# EPICS substitutions: pmacApp/Db/pmac.substitutions
# This file was automatically generated on Thu 15 Nov 2018 14:28:58 GMT from
# source: /home/hgv27681/R3.14.12.7/support/pmac/etc/makeIocs/lab.xml
#
# *** Please do not edit this file: edit the source file instead. ***
#

# Macros:
#  PORT      The asyn port for the pmac controller
#  P         PV Prefix
#  NAXES     Number of axes
#  TIMEOUT   Timeout for controller communication
#  FEEDRATE  feedrate below which we go into error
#  CSG0      Name for Coordinate System Group 0
#  CSG1      Name for Coordinate System Group 1
#  CSG2      Name for Coordinate System Group 2
#  CSG3      Name for Coordinate System Group 3
#  CSG4      Name for Coordinate System Group 4
#  CSG5      Name for Coordinate System Group 5
#  CSG6      Name for Coordinate System Group 6
#  CSG7      Name for Coordinate System Group 7
#file /usr/local/epics-nfs/apps/pmac/2019_05_14_01/db/pmacController.template
file /usr/local/epics-nfs/apps/pmac/pmacApp/Db/pmacController.template
{
pattern { PORT, P, NAXES, TIMEOUT, FEEDRATE, CSG0, CSG1, CSG2, CSG3, CSG4, CSG5, CSG6, CSG7 }
    { "Brick", "BRICK1", "8", "4", "100", "", "", "", "", "", "", "", "" }
}

# Macros:
#  PORT  The asyn port for the pmac controller
#  P     PV Prefix
#file /usr/local/epics-nfs/apps/pmac/2019_05_14_01/db/powerPmacStatus.template
file /usr/local/epics-nfs/apps/pmac/pmacApp/Db/powerPmacStatus.template
{
pattern { PORT, P }
    { "Brick", "BRICK1" }
}

# Macros:
#  PMAC  Pmac/Geobrick name
#  AXIS  Axis number
#  PORT  Asyn port
#file /usr/local/epics-nfs/apps/pmac/2019_05_14_01/db/pmacStatusAxis.template
file /usr/local/epics-nfs/apps/pmac/pmacApp/Db/pmacStatusAxis.template
{
pattern { PMAC, AXIS, PORT }
    { "BRICK1", "1", "Brick" }
    { "BRICK1", "2", "Brick" }
    { "BRICK1", "3", "Brick" }
    { "BRICK1", "4", "Brick" }
    { "BRICK1", "5", "Brick" }
    { "BRICK1", "6", "Brick" }
    { "BRICK1", "7", "Brick" }
    { "BRICK1", "8", "Brick" }
}

#file /usr/local/epics-nfs/apps/pmac/2019_05_14_01/db/pmacCsController.template
#{
#pattern {PORT, PARENTPORT, TIMEOUT, PMAC, CS}
#	{"CS1", "Brick", 100, "BRICK1", 1}
#}

# Macros:
#  P           Device Prefix
#  M           Device Suffix
#  PORT        Delta tau motor CS
#  ADDR        Address on controller
#  DESC        Description, displayed on EDM screen
#  MRES        Motor Step Size (EGU)
#  VELO        Velocity (EGU/s)
#  PREC        Display Precision
#  EGU         Engineering Units
#  TWV         Tweak Step Size (EGU)
#  DTYP        DTYP of record
#  DIR         User Direction
#  VBAS        Base Velocity (EGU/s)
#  VMAX        Max Velocity (EGU/s), defaults to VELO
#  ACCL        Seconds to Velocity
#  BDST        BL Distance (EGU)
#  BVEL        BL Velocity (EGU/s)
#  BACC        BL Seconds to Veloc.
#  DHLM        Dial High Limit
#  DLLM        Dial Low Limit
#  HLM         User High Limit
#  LLM         User Low Limit
#  HLSV        HW Lim. Violation Svr
#  INIT        Startup commands
#  SREV        Steps per Revolution
#  RRES        Readback Step Size (EGU)
#  ERES        Encoder Step Size (EGU)
#  JAR         Jog Acceleration (EGU/s^2)
#  UEIP        Use Encoder If Present
#  URIP        Use RDBL If Present
#  RDBL        Readback Location, set URIP = 1 if you specify this
#  RTRY        Max retry count
#  DLY         Readback settle time (s)
#  OFF         User Offset (EGU)
#  RDBD        Retry Deadband (EGU)
#  FOFF        Freeze Offset, 0=variable, 1=frozen
#  ADEL        Alarm monitor deadband (EGU)
#  NTM         New Target Monitor, only set to 0 for soft motors
#  FEHIGH      HIGH limit for following error
#  FEHIHI      HIHI limit for following error
#  FEHHSV      HIHI alarm severity for following error
#  FEHSV       HIGH alarm severity for following error
#  SCALE       Scale factor, if pmacSetAxisScale is used this should be set
#  HOMEVIS     If 1 then home is visible on the gui
#  HOMEVISSTR  If HOMEVIS=0, then display this text on the gui instead
#  name        Object name and gui association name
#  alh         Set this to alh to add the motor to the alarm handler and send emails,
#  gda_name    Name to export this as to GDA
#  gda_desc    Description to export this as to GDA
#  HOME        Prefix for autohome instance. Defaults to $(P). If unspecified,
#file /usr/local/epics-nfs/apps/pmac/2019_05_14_01/db/dls_pmac_cs_asyn_motor.template
file /usr/local/epics-nfs/apps/pmac/pmacApp/Db/dls_pmac_cs_asyn_motor.template
{
pattern { P, M, PORT, ADDR, DESC, MRES, VELO, PREC, EGU, TWV, DTYP, DIR, VBAS, VMAX, ACCL, BDST, BVEL, BACC, DHLM, DLLM, HLM, LLM, HLSV, INIT, SREV, RRES, ERES, JAR, UEIP, URIP, RDBL, RTRY, DLY, OFF, RDBD, FOFF, ADEL, NTM, FEHIGH, FEHIHI, FEHHSV, FEHSV, SCALE, HOMEVIS, HOMEVISSTR, name, alh, gda_name, gda_desc, HOME, PMAC, CS }
  { "BL", ":vm1", "CS1", "1", "Test motor", "1", "100", "3", "mm", "0.0", "asynMotor", "0", "0", "1000", "0.5", "0", "0", "", "", "", "", "", "MAJOR", "", "1000", "", "", "", "0", "0", "", "0", "0", "0", "", "0", "0", "1", "0", "0", "NO_ALARM", "NO_ALARM", "1", "1", "Use motor summary screen", "BRICK1.MOTORS.M1", "None", "", "Test", "$(P)", "BRICK1", "1" }
  { "BL", ":vm2", "CS1", "2", "Test motor", "1", "100", "3", "mm", "0.0", "asynMotor", "0", "0", "1000", "0.5", "0", "0", "", "", "", "", "", "MAJOR", "", "1000", "", "", "", "0", "0", "", "0", "0", "0", "", "0", "0", "1", "0", "0", "NO_ALARM", "NO_ALARM", "1", "1", "Use motor summary screen", "BRICK1.MOTORS.M2", "None", "", "Test", "$(P)", "BRICK1", "1" }
  { "BL", ":vm3", "CS1", "3", "Test motor", "1", "100", "3", "mm", "0.0", "asynMotor", "0", "0", "1000", "0.5", "0", "0", "", "", "", "", "", "MAJOR", "", "1000", "", "", "", "0", "0", "", "0", "0", "0", "", "0", "0", "1", "0", "0", "NO_ALARM", "NO_ALARM", "1", "1", "Use motor summary screen", "BRICK1.MOTORS.M3", "None", "", "Test", "$(P)", "BRICK1", "1" }
  { "BL", ":vm5", "CS1", "5", "Test motor", "1", "100", "3", "mm", "0.0", "asynMotor", "0", "0", "1000", "0.5", "0", "0", "", "", "", "", "", "MAJOR", "", "1000", "", "", "", "0", "0", "", "0", "0", "0", "", "0", "0", "1", "0", "0", "NO_ALARM", "NO_ALARM", "1", "1", "Use motor summary screen", "BRICK1.MOTORS.M5", "None", "", "Test", "$(P)", "BRICK1", "1" }
  { "BL", ":vm6", "CS1", "6", "Test motor", "1", "100", "3", "mm", "0.0", "asynMotor", "0", "0", "1000", "0.5", "0", "0", "", "", "", "", "", "MAJOR", "", "1000", "", "", "", "0", "0", "", "0", "0", "0", "", "0", "0", "1", "0", "0", "NO_ALARM", "NO_ALARM", "1", "1", "Use motor summary screen", "BRICK1.MOTORS.M6", "None", "", "Test", "$(P)", "BRICK1", "1" }
  { "BL", ":Gap", "CS1", "7", "Horizontal gap", "0.048828125", "10", "3", "um", "0.0", "asynMotor", "0", "0", "1000", "0.5", "0", "0", "", "10000", "-10000", "10000", "-10000", "MAJOR", "", "8192", "", "", "", "0", "0", "", "0", "0", "0", "", "0", "0", "1", "0", "0", "NO_ALARM", "NO_ALARM", "1", "1", "Use motor summary screen", "BRICK1.MOTORS.M7", "None", "", "Test", "$(P)", "BRICK1", "1" }
  { "BL", ":Offset", "CS1", "8", "Horizontal offset", "0.048828125", "10", "3", "um", "0.0", "asynMotor", "0", "0", "1000", "0.5", "0", "0", "", "10000", "-10000", "10000", "-10000", "MAJOR", "", "8192", "", "", "", "0", "0", "", "0", "0", "0", "", "0", "0", "1", "0", "0", "NO_ALARM", "NO_ALARM", "1", "1", "Use motor summary screen", "BRICK1.MOTORS.M8", "None", "", "Test", "$(P)", "BRICK1", "1" }
  { "BL", ":Gap", "CS2", "7", "Vertical gap", "0.048828125", "10", "3", "um", "0.0", "asynMotor", "0", "0", "1000", "0.5", "0", "0", "", "10000", "-10000", "10000", "-10000", "MAJOR", "", "8192", "", "", "", "0", "0", "", "0", "0", "0", "", "0", "0", "1", "0", "0", "NO_ALARM", "NO_ALARM", "1", "1", "Use motor summary screen", "BRICK1.MOTORS.M7", "None", "", "Test", "$(P)", "BRICK1", "2" }
  { "BL", ":Offset", "CS2", "8", "Vertical offset", "0.048828125", "10", "3", "um", "0.0", "asynMotor", "0", "0", "1000", "0.5", "0", "0", "", "10000", "-10000", "10000", "-10000", "MAJOR", "", "8192", "", "", "", "0", "0", "", "0", "0", "0", "", "0", "0", "1", "0", "0", "NO_ALARM", "NO_ALARM", "1", "1", "Use motor summary screen", "BRICK1.MOTORS.M8", "None", "", "Test", "$(P)", "BRICK1", "2" }
}

# Macros:
#  P                Device Prefix
#  M                Device Suffix
#  PORT             Delta tau motor controller
#  ADDR             Address on controller
#  DESC             Description, displayed on EDM screen
#  MRES             Motor Step Size (EGU)
#  VELO             Velocity (EGU/s)
#  PREC             Display Precision
#  EGU              Engineering Units
#  TWV              Tweak Step Size (EGU)
#  DTYP             DTYP of record
#  DIR              User Direction
#  VBAS             Base Velocity (EGU/s)
#  VMAX             Max Velocity (EGU/s), defaults to VELO
#  ACCL             Seconds to Velocity
#  BDST             BL Distance (EGU)
#  BVEL             BL Velocity (EGU/s)
#  BACC             BL Seconds to Veloc.
#  DHLM             Dial High Limit
#  DLLM             Dial Low Limit
#  HLM              User High Limit
#  LLM              User Low Limit
#  HLSV             HW Lim. Violation Svr
#  INIT             Startup commands
#  SREV             Steps per Revolution
#  RRES             Readback Step Size (EGU)
#  ERES             Encoder Step Size (EGU)
#  JAR              Jog Acceleration (EGU/s^2)
#  UEIP             Use Encoder If Present
#  URIP             Use RDBL If Present
#  RDBL             Readback Location, set URIP = 1 if you specify this
#  RTRY             Max retry count
#  DLY              Readback settle time (s)
#  OFF              User Offset (EGU)
#  RDBD             Retry Deadband (EGU)
#  FOFF             Freeze Offset, 0=variable, 1=frozen
#  ADEL             Alarm monitor deadband (EGU)
#  NTM              New Target Monitor, only set to 0 for soft motors
#  FEHIGH           HIGH limit for following error
#  FEHIHI           HIHI limit for following error
#  FEHHSV           HIHI alarm severity for following error
#  FEHSV            HIGH alarm severity for following error
#  SCALE            Scale factor, if pmacSetAxisScale is used this should be set
#  HOMEVIS          If 1 then home is visible on the gui
#  HOMEVISSTR       If HOMEVIS=0, then display this text on the gui instead
#  name             Object name and gui association name
#  alh              Set this to alh to add the motor to the alarm handler and send emails,
#  gda_name         Name to export this as to GDA
#  gda_desc         Description to export this as to GDA
#  SPORT            Delta tau motor controller comms port
#  HOME             Prefix for autohome instance. Defaults to $(P). If unspecified,
#  PMAC             Prefix for pmacStatus instance. Needed to get axis descriptions
#  ALLOW_HOMED_SET  Set to a blank to allow this axis to have its homed
#file /usr/local/epics-nfs/apps/pmac/2019_05_14_01/db/dls_pmac_asyn_motor.template
file /usr/local/epics-nfs/apps/pmac/pmacApp/Db/dls_pmac_asyn_motor.template
{
pattern { P, M, PORT, ADDR, DESC, MRES, VELO, PREC, EGU, TWV, DTYP, DIR, VBAS, VMAX, ACCL, BDST, BVEL, BACC, DHLM, DLLM, HLM, LLM, HLSV, INIT, SREV, RRES, ERES, JAR, UEIP, URIP, RDBL, RTRY, DLY, OFF, RDBD, FOFF, ADEL, NTM, FEHIGH, FEHIHI, FEHHSV, FEHSV, SCALE, HOMEVIS, HOMEVISSTR, name, alh, gda_name, gda_desc, SPORT, HOME, PMAC, ALLOW_HOMED_SET }
  { "BL", ":m1", "Brick", "1", "Right", "0.048828125", "10", "3", "um", "1", "asynMotor", "0", "0", "1000", "0.5", "0", "0", "", "0", "0", "", "", "MAJOR", "", "8192", "", "", "", "0", "0", "", "0", "0", "0", "", "0", "0", "1", "0", "0", "NO_ALARM", "NO_ALARM", "1", "1", "Use motor summary screen", "BRICK1.MOTORS.M1", "None", "", "Test", "BRICK1port", "$(P)", "BRICK1", "#" }
  { "BL", ":m2", "Brick", "2", "Left", "0.048828125", "10", "3", "um", "1", "asynMotor", "0", "0", "1000", "0.5", "0", "0", "", "10000", "-10000", "10000", "-10000", "MAJOR", "", "8192", "", "", "", "0", "0", "", "0", "0", "0", "", "0", "0", "1", "0", "0", "NO_ALARM", "NO_ALARM", "1", "1", "Use motor summary screen", "BRICK1.MOTORS.M2", "None", "", "Test", "BRICK1port", "$(P)", "BRICK1", "#" }
  { "BL", ":m3", "Brick", "3", "Top", "0.048828125", "10", "3", "um", "1", "asynMotor", "0", "0", "1000", "0.5", "0", "0", "", "0", "0", "", "", "MAJOR", "", "8192", "", "", "", "0", "0", "", "0", "0", "0", "", "0", "0", "1", "0", "0", "NO_ALARM", "NO_ALARM", "1", "1", "Use motor summary screen", "BRICK1.MOTORS.M3", "None", "", "Test", "BRICK1port", "$(P)", "BRICK1", "#" }
  { "BL", ":m4", "Brick", "4", "Bottom", "0.048828125", "10", "3", "um", "1", "asynMotor", "0", "0", "1000", "0.5", "0", "0", "", "10000", "-10000", "10000", "-10000", "MAJOR", "", "8192", "", "", "", "0", "0", "", "0", "0", "0", "", "0", "0", "1", "0", "0", "NO_ALARM", "NO_ALARM", "1", "1", "Use motor summary screen", "BRICK1.MOTORS.M4", "None", "", "Test", "BRICK1port", "$(P)", "BRICK1", "#" }
  { "BL", ":m5", "Brick", "5", "Motor 5", "1", "100", "3", "mm", "1", "asynMotor", "0", "0", "1000", "0.5", "0", "0", "", "0", "0", "", "", "MAJOR", "", "1000", "", "", "", "0", "0", "", "0", "0", "0", "", "0", "0", "1", "0", "0", "NO_ALARM", "NO_ALARM", "1", "1", "Use motor summary screen", "BRICK1.MOTORS.M5", "None", "", "Test", "BRICK1port", "$(P)", "BRICK1", "#" }
  { "BL", ":m6", "Brick", "6", "Motor 6", "1", "100", "3", "mm", "1", "asynMotor", "0", "0", "1000", "0.5", "0", "0", "", "0", "0", "", "", "MAJOR", "", "1000", "", "", "", "0", "0", "", "0", "0", "0", "", "0", "0", "1", "0", "0", "NO_ALARM", "NO_ALARM", "1", "1", "Use motor summary screen", "BRICK1.MOTORS.M6", "None", "", "Test", "BRICK1port", "$(P)", "BRICK1", "#" }
  { "BL", ":m7", "Brick", "7", "Motor 7", "1", "100", "3", "mm", "1", "asynMotor", "0", "0", "1000", "0.5", "0", "0", "", "0", "0", "", "", "MAJOR", "", "1000", "", "", "", "0", "0", "", "0", "0", "0", "", "0", "0", "1", "0", "0", "NO_ALARM", "NO_ALARM", "1", "1", "Use motor summary screen", "BRICK1.MOTORS.M7", "None", "", "Test", "BRICK1port", "$(P)", "BRICK1", "#" }
  { "BL", ":m8", "Brick", "8", "Motor 8", "1", "100", "3", "mm", "1", "asynMotor", "0", "0", "1000", "0.5", "0", "0", "", "0", "0", "", "", "MAJOR", "", "1000", "", "", "", "0", "0", "", "0", "0", "0", "", "0", "0", "1", "0", "0", "NO_ALARM", "NO_ALARM", "1", "1", "Use motor summary screen", "BRICK1.MOTORS.M8", "None", "", "Test", "BRICK1port", "$(P)", "BRICK1", "#" }
}
